binaryValueToTest := ADR(valueToTest);
assertionIsWrong := (binaryValueToTest^ <> THIS^.BINARY_NEGATIVE_INFINITY);

message := SEL(
	assertionIsWrong,
	'currentValue is %s assertion must be TRUE', 
	'currentValue is %s assertion must be FALSE'
);

valueToTestAsString := TO_STRING(valueToTest);

messageStringBuilder(
	sFormat := message,
	arg1 := THIS^.AnyToArg(valueToTestAsString)
);

THIS^.assertorContainer.assertor.assert.float.single.valueIsNegativeInfinite(
	currentValue := valueToTest,
	message := ''
);

THIS^.AssertEquals_BOOL(
	Expected 	:= assertionIsWrong,
	Actual 		:= THIS^.assertorContainer.wasAssertionWrong,
	Message 	:= messageStringBuilder.sOut
);
END_METHOD

(*

short summary
==================
This test method tests ``assert.float.single.valueIsNegativeZero``
method of CNM_AssertionInterfaces library, 
it provides the possibility to handover test data via parameter 

.. <legal notes>

legal notes
=================
| SPDX-FileCopyrightText: © 2022 ekvip automation GmbH <info@ekvip.de>
| SPDX-License-Identifier: Apache-2.0
| For details check: Apache-2.0_

.. _Apache-2.0: https://www.apache.org/licenses/LICENSE-2.0

.. </legal notes>

parameters
==========

*)

METHOD testValueIsNegativeZero
VAR_INPUT
	(* for the test it's the parameter ``currentValue`` *)
	valueToTest	:REAL;	
END_VAR
VAR
	(* just the expectation if the assertion to test must be worng or true *)
	assertionIsWrong		:BOOL;
	(* contains the format string for the test message *)
	message					:Tc2_System.T_MaxString;
	(* TwinCAT printf with the test message *)
	messageStringBuilder	:Tc2_Utilities.FB_FormatString;
	(* value of the paramter ``valueToTest`` as string *)
	valueToTestAsString		:Tc2_System.T_MaxString;
	(* binary value of the parameter ``valueToTest`` *)
	binaryValueToTest		:POINTER TO DWORD;
	(* sgin bit as BYTE for the message *)
	signBitAsByte			:BYTE;
	(* sgin bit as BOOL for the message *)
	signBit					:BOOL;	
END_VAR
THIS^.assertorContainer.resetAssertor();

binaryValueToTest := ADR(valueToTest);
signBit := binaryValueToTest^.SIGN;
signBitAsByte := TO_BYTE(signBit);

assertionIsWrong := (binaryValueToTest^ <> THIS^.BINARY_MINUS_ZERO);

message := SEL(
	assertionIsWrong,
	'currentValue is %s and sign bit is %u assertion must be TRUE', 
	'currentValue is %s and sign bit is %u assertion must be FALSE'
);

valueToTestAsString := TO_STRING(valueToTest);

messageStringBuilder(
	sFormat := message,
	arg1 := THIS^.AnyToArg(valueToTestAsString),
	arg2 := THIS^.AnyToArg(signBitAsByte)
);

THIS^.assertorContainer.assertor.assert.float.single.valueIsNegativeZero(
	currentValue := valueToTest,
	message := ''
);

THIS^.AssertEquals_BOOL(
	Expected 	:= assertionIsWrong,
	Actual 		:= THIS^.assertorContainer.wasAssertionWrong,
	Message 	:= messageStringBuilder.sOut
);
END_METHOD

(*

short summary
==================
This test method tests ``assert.float.single.valueIsNormal``
method of CNM_AssertionInterfaces library, 
it provides the possibility to handover test data via parameter 

.. <legal notes>

legal notes
=================
| SPDX-FileCopyrightText: © 2022 ekvip automation GmbH <info@ekvip.de>
| SPDX-License-Identifier: Apache-2.0
| For details check: Apache-2.0_

.. _Apache-2.0: https://www.apache.org/licenses/LICENSE-2.0

.. </legal notes>

parameters
==========

*)

METHOD testValueIsNormal
VAR_INPUT
	(* for the test it's the parameter ``currentValue`` *)
	valueToTest	:REAL;	
END_VAR
VAR
	(* just the expectation if the assertion to test must be worng or true *)
	assertionIsWrong		:BOOL;
	(* contains the format string for the test message *)
	message					:Tc2_System.T_MaxString;
	(* TwinCAT printf with the test message *)
	messageStringBuilder	:Tc2_Utilities.FB_FormatString;
	(* value of the paramter ``valueToTest`` as string *)
	valueToTestAsString		:Tc2_System.T_MaxString;
	(* binary value of the parameter ``valueToTest`` *)
	binaryValueToTest		:POINTER TO DWORD;
END_VAR
THIS^.assertorContainer.resetAssertor();

binaryValueToTest := ADR(valueToTest);

assertionIsWrong := (
	((binaryValueToTest^ AND THIS^.MASK_FOR_EXPONENT) = THIS^.BINARY_ZERO)
	OR_ELSE Tc2_Utilities.RealIsNaN(valueToTest)
	OR_ELSE (NOT Tc2_Utilities.RealIsFinite(valueToTest))
);

message := SEL(
	assertionIsWrong,
	'currentValue is %s assertion must be TRUE', 
	'currentValue is %s assertion must be FALSE'
);

valueToTestAsString := TO_STRING(valueToTest);

messageStringBuilder(
	sFormat := message,
	arg1 := THIS^.AnyToArg(valueToTestAsString)
);

THIS^.assertorContainer.assertor.assert.float.single.valueIsNormal(
	currentValue := valueToTest,
	message := ''
);

THIS^.AssertEquals_BOOL(
	Expected 	:= assertionIsWrong,
	Actual 		:= THIS^.assertorContainer.wasAssertionWrong,
	Message 	:= messageStringBuilder.sOut
);
END_METHOD

(*

short summary
==================
This test method tests ``assert.float.single.valueIsNotEqualTo``
method of CNM_AssertionInterfaces library, 
it provides the possibility to handover test data via parameter 


.. <legal notes>

legal notes
=================
| SPDX-FileCopyrightText: © 2022 ekvip automation GmbH <info@ekvip.de>
| SPDX-License-Identifier: Apache-2.0
| For details check: Apache-2.0_

.. _Apache-2.0: https://www.apache.org/licenses/LICENSE-2.0

.. </legal notes>

parameters
==========

*)

METHOD testValueIsNotEqualTo 
VAR_INPUT
	(* for the test it's the parameter ``currentValue`` *)
	valueToTest		:REAL;
	(* for the test it's the parameter ``unexpectedValue`` *)
	unexpectedValue	:REAL;
	(* for the test it's the parameter ``tolerance`` *)
	tolerance		:REAL;
END_VAR
VAR
	(* just the expectation if the assertion to test must be worng or true *)
	assertionIsWrong		:BOOL;
	(* contains the format string for the test message *)
	message					:Tc2_System.T_MaxString;
	(* TwinCAT printf with the test message *)
	messageStringBuilder	:Tc2_Utilities.FB_FormatString;
	(* just to cast *)
	binaryCurrentValue		:POINTER TO DWORD;
	(* just to cast *)
	binaryUnexpectedValue	:POINTER TO DWORD;
	(* value of the paramter ``valueToTest`` as string *)
	valueToTestAsString		:Tc2_System.T_MaxString;
	(* value of the paramter ``unexpectedValue`` as string *)
	unexpectedValueAsString	:Tc2_System.T_MaxString;
	(* value of the paramter ``tolerance`` as string *)
	toleranceAsString		:Tc2_System.T_MaxString;	
END_VAR
THIS^.assertorContainer.resetAssertor();
IF (
	Tc2_Utilities.RealIsNaN(valueToTest)
	OR Tc2_Utilities.RealIsNaN(unexpectedValue)
	OR Tc2_Utilities.RealIsNaN(tolerance)
) THEN
	assertionIsWrong := FALSE;
ELSIF (NOT Tc2_Utilities.RealIsFinite(tolerance)) THEN
	assertionIsWrong := TRUE;
ELSIF (Tc2_Utilities.RealIsFinite(valueToTest) <> Tc2_Utilities.RealIsFinite(unexpectedValue)) THEN
	assertionIsWrong := FALSE; 
ELSIF (
	(NOT Tc2_Utilities.RealIsFinite(valueToTest))
	OR (NOT Tc2_Utilities.RealIsFinite(unexpectedValue))
) THEN
	binaryCurrentValue := ADR(valueToTest);
	binaryUnexpectedValue := ADR(unexpectedValue);
	assertionIsWrong := (binaryCurrentValue^.SIGN = binaryUnexpectedValue^.SIGN);
ELSE
	assertionIsWrong := (
		((unexpectedValue + ABS(tolerance)) >= valueToTest)
		AND ((unexpectedValue - ABS(tolerance)) <= valueToTest)
	);
END_IF

message := SEL(
	assertionIsWrong,
	'currentValue is %s unexpectedValue is %s tolerance is %s assertion must be TRUE', 
	'currentValue is %s unexpectedValue is %s tolerance is %s assertion must be FALSE'
);

valueToTestAsString := TO_STRING(valueToTest);
unexpectedValueAsString := TO_STRING(unexpectedValue);
toleranceAsString := TO_STRING(tolerance);

messageStringBuilder(
	sFormat := message,
	arg1 := THIS^.AnyToArg(valueToTestAsString),
	arg2 := THIS^.AnyToArg(unexpectedValueAsString),
	arg3 := THIS^.AnyToArg(toleranceAsString)
);

THIS^.assertorContainer.assertor.assert.float.single.valueIsNotEqualTo(
	currentValue	:= valueToTest,
	unexpectedValue	:= unexpectedValue,
	tolerance       := tolerance,
	message			:= ''
);

THIS^.AssertEquals_BOOL(
	Expected 	:= assertionIsWrong,
	Actual 		:= THIS^.assertorContainer.wasAssertionWrong,
	Message 	:= messageStringBuilder.sOut
);
END_METHOD

(*

short summary
==================
This test method tests ``assert.float.single.valueIsNotNegativeInfinite``
method of CNM_AssertionInterfaces library, 
it provides the possibility to handover test data via parameter 

.. <legal notes>

legal notes
=================
| SPDX-FileCopyrightText: © 2022 ekvip automation GmbH <info@ekvip.de>
| SPDX-License-Identifier: Apache-2.0
| For details check: Apache-2.0_

.. _Apache-2.0: https://www.apache.org/licenses/LICENSE-2.0

.. </legal notes>

parameters
==========

*)

METHOD testValueIsNotNegativeInfinite
VAR_INPUT
	(* for the test it's the parameter ``currentValue`` *)
	valueToTest	:REAL;	
END_VAR
VAR
	(* just the expectation if the assertion to test must be worng or true *)
	assertionIsWrong		:BOOL;
	(* contains the format string for the test message *)
	message					:Tc2_System.T_MaxString;
	(* TwinCAT printf with the test message *)
	messageStringBuilder	:Tc2_Utilities.FB_FormatString;
	(* value of the paramter ``valueToTest`` as string *)
	valueToTestAsString		:Tc2_System.T_MaxString;
	(* binary value of the parameter ``valueToTest`` *)
	binaryValueToTest		:POINTER TO DWORD;
END_VAR
THIS^.assertorContainer.resetAssertor();

binaryValueToTest := ADR(valueToTest);
assertionIsWrong := (binaryValueToTest^ = THIS^.BINARY_NEGATIVE_INFINITY);

message := SEL(
	assertionIsWrong,
	'currentValue is %s assertion must be TRUE', 
	'currentValue is %s assertion must be FALSE'
);

valueToTestAsString := TO_STRING(valueToTest);

messageStringBuilder(
	sFormat := message,
	arg1 := THIS^.AnyToArg(valueToTestAsString)
);

THIS^.assertorContainer.assertor.assert.float.single.valueIsNotNegativeInfinite(
	currentValue := valueToTest,
	message := ''
);

THIS^.AssertEquals_BOOL(
	Expected 	:= assertionIsWrong,
	Actual 		:= THIS^.assertorContainer.wasAssertionWrong,
	Message 	:= messageStringBuilder.sOut
);
END_METHOD

(*

short summary
==================
This test method tests ``assert.float.single.valueIsNotPositiveInfinite``
method of CNM_AssertionInterfaces library, 
it provides the possibility to handover test data via parameter 

.. <legal notes>

legal notes
=================
| SPDX-FileCopyrightText: © 2022 ekvip automation GmbH <info@ekvip.de>
| SPDX-License-Identifier: Apache-2.0
| For details check: Apache-2.0_

.. _Apache-2.0: https://www.apache.org/licenses/LICENSE-2.0

.. </legal notes>

parameters
==========

*)

METHOD testValueIsNotPositiveInfinite
VAR_INPUT
	(* for the test it's the parameter ``currentValue`` *)
	valueToTest	:REAL;	
END_VAR
VAR
	(* just the expectation if the assertion to test must be worng or true *)
	assertionIsWrong		:BOOL;
	(* contains the format string for the test message *)
	message					:Tc2_System.T_MaxString;
	(* TwinCAT printf with the test message *)
	messageStringBuilder	:Tc2_Utilities.FB_FormatString;
	(* value of the paramter ``valueToTest`` as string *)
	valueToTestAsString		:Tc2_System.T_MaxString;
	(* binary value of the parameter ``valueToTest`` *)
	binaryValueToTest		:POINTER TO DWORD;
END_VAR
THIS^.assertorContainer.resetAssertor();

binaryValueToTest := ADR(valueToTest);
assertionIsWrong := (binaryValueToTest^ = THIS^.BINARY_INFINITY);

message := SEL(
	assertionIsWrong,
	'currentValue is %s assertion must be TRUE', 
	'currentValue is %s assertion must be FALSE'
);

valueToTestAsString := TO_STRING(valueToTest);

messageStringBuilder(
	sFormat := message,
	arg1 := THIS^.AnyToArg(valueToTestAsString)
);

THIS^.assertorContainer.assertor.assert.float.single.valueIsNotPositiveInfinite(
	currentValue := valueToTest,
	message := ''
);

THIS^.AssertEquals_BOOL(
	Expected 	:= assertionIsWrong,
	Actual 		:= THIS^.assertorContainer.wasAssertionWrong,
	Message 	:= messageStringBuilder.sOut
);
END_METHOD

(*

short summary
==================
This test method tests ``assert.float.single.valueIsNotSpecial``
method of CNM_AssertionInterfaces library, 
it provides the possibility to handover test data via parameter 

.. <legal notes>

legal notes
=================
| SPDX-FileCopyrightText: © 2022 ekvip automation GmbH <info@ekvip.de>
| SPDX-License-Identifier: Apache-2.0
| For details check: Apache-2.0_

.. _Apache-2.0: https://www.apache.org/licenses/LICENSE-2.0

.. </legal notes>

parameters
==========

*)

METHOD testValueIsNotSpecial
VAR_INPUT
	(* for the test it's the parameter ``currentValue`` *)
	valueToTest	:REAL;	
END_VAR
VAR
	(* just the expectation if the assertion to test must be worng or true *)
	assertionIsWrong		:BOOL;
	(* contains the format string for the test message *)
	message					:Tc2_System.T_MaxString;
	(* TwinCAT printf with the test message *)
	messageStringBuilder	:Tc2_Utilities.FB_FormatString;
	(* value of the paramter ``valueToTest`` as string *)
	valueToTestAsString		:Tc2_System.T_MaxString;
END_VAR
THIS^.assertorContainer.resetAssertor();

assertionIsWrong := (
	(NOT Tc2_Utilities.RealIsFinite(valueToTest))
	OR_ELSE Tc2_Utilities.RealIsNaN(valueToTest)
);

message := SEL(
	assertionIsWrong,
	'currentValue is %s assertion must be TRUE', 
	'currentValue is %s assertion must be FALSE'
);

valueToTestAsString := TO_STRING(valueToTest);

messageStringBuilder(
	sFormat := message,
	arg1 := THIS^.AnyToArg(valueToTestAsString)
);

THIS^.assertorContainer.assertor.assert.float.single.valueIsNotSpecial(
	currentValue := valueToTest,
	message := ''
);

THIS^.AssertEquals_BOOL(
	Expected 	:= assertionIsWrong,
	Actual 		:= THIS^.assertorContainer.wasAssertionWrong,
	Message 	:= messageStringBuilder.sOut
);
END_METHOD

(*

short summary
==================
This test method tests ``assert.float.single.valueIsPositive``
method of CNM_AssertionInterfaces library, 
it provides the possibility to handover test data via parameter 

.. <legal notes>

legal notes
=================
| SPDX-FileCopyrightText: © 2022 ekvip automation GmbH <info@ekvip.de>
| SPDX-License-Identifier: Apache-2.0
| For details check: Apache-2.0_

.. _Apache-2.0: https://www.apache.org/licenses/LICENSE-2.0

.. </legal notes>

parameters
==========

*)

METHOD testValueIsPositive
VAR_INPUT
	(* for the test it's the parameter ``currentValue`` *)
	valueToTest	:REAL;	
END_VAR
VAR
	(* just the expectation if the assertion to test must be worng or true *)
	assertionIsWrong		:BOOL;
	(* contains the format string for the test message *)
	message					:Tc2_System.T_MaxString;
	(* TwinCAT printf with the test message *)
	messageStringBuilder	:Tc2_Utilities.FB_FormatString;
	(* value of the paramter ``valueToTest`` as string *)
	valueToTestAsString		:Tc2_System.T_MaxString;
	(* binary value of the parameter ``valueToTest`` *)
	binaryValueToTest		:POINTER TO DWORD;
	(* sgin bit as BYTE for the message *)
	signBitAsByte			:BYTE;
	(* sgin bit as BOOL for the message *)
	signBit					:BOOL;	
END_VAR
THIS^.assertorContainer.resetAssertor();

binaryValueToTest := ADR(valueToTest);
signBit := binaryValueToTest^.SIGN;
signBitAsByte := TO_BYTE(signBit);
assertionIsWrong := (
	signBit
	OR Tc2_Utilities.RealIsNaN(valueToTest)
);

message := SEL(
	assertionIsWrong,
	'currentValue is %s and sign bit is %u assertion must be TRUE', 
	'currentValue is %s and sign bit is %u assertion must be FALSE'
);

valueToTestAsString := TO_STRING(valueToTest);

messageStringBuilder(
	sFormat := message,
	arg1 := THIS^.AnyToArg(valueToTestAsString),
	arg2 := THIS^.AnyToArg(signBitAsByte)
);

THIS^.assertorContainer.assertor.assert.float.single.valueIsPositive(
	currentValue := valueToTest,
	message := ''
);

THIS^.AssertEquals_BOOL(
	Expected 	:= assertionIsWrong,
	Actual 		:= THIS^.assertorContainer.wasAssertionWrong,
	Message 	:= messageStringBuilder.sOut
);
END_METHOD

(*

short summary
==================
This test method tests ``assert.float.single.valueIsPositiveInfinite``
method of CNM_AssertionInterfaces library, 
it provides the possibility to handover test data via parameter 

.. <legal notes>

legal notes
=================
| SPDX-FileCopyrightText: © 2022 ekvip automation GmbH <info@ekvip.de>
| SPDX-License-Identifier: Apache-2.0
| For details check: Apache-2.0_

.. _Apache-2.0: https://www.apache.org/licenses/LICENSE-2.0

.. </legal notes>

parameters
==========

*)

METHOD testValueIsPositiveInfinite
VAR_INPUT
	(* for the test it's the parameter ``currentValue`` *)
	valueToTest	:REAL;	
END_VAR
VAR
	(* just the expectation if the assertion to test must be worng or true *)
	assertionIsWrong		:BOOL;
	(* contains the format string for the test message *)
	message					:Tc2_System.T_MaxString;
	(* TwinCAT printf with the test message *)
	messageStringBuilder	:Tc2_Utilities.FB_FormatString;
	(* value of the paramter ``valueToTest`` as string *)
	valueToTestAsString		:Tc2_System.T_MaxString;
	(* binary value of the parameter ``valueToTest`` *)
	binaryValueToTest		:POINTER TO DWORD;
END_VAR
THIS^.assertorContainer.resetAssertor();

binaryValueToTest := ADR(valueToTest);
assertionIsWrong := (binaryValueToTest^ <> THIS^.BINARY_INFINITY);

message := SEL(
	assertionIsWrong,
	'currentValue is %s assertion must be TRUE', 
	'currentValue is %s assertion must be FALSE'
);

valueToTestAsString := TO_STRING(valueToTest);

messageStringBuilder(
	sFormat := message,
	arg1 := THIS^.AnyToArg(valueToTestAsString)
);

THIS^.assertorContainer.assertor.assert.float.single.valueIsPositiveInfinite(
	currentValue := valueToTest,
	message := ''
);

THIS^.AssertEquals_BOOL(
	Expected 	:= assertionIsWrong,
	Actual 		:= THIS^.assertorContainer.wasAssertionWrong,
	Message 	:= messageStringBuilder.sOut
);
END_METHOD

(*

short summary
==================
This test method tests ``assert.float.single.valueIsPositiveZero``
method of CNM_AssertionInterfaces library, 
it provides the possibility to handover test data via parameter 

.. <legal notes>

legal notes
=================
| SPDX-FileCopyrightText: © 2022 ekvip automation GmbH <info@ekvip.de>
| SPDX-License-Identifier: Apache-2.0
| For details check: Apache-2.0_

.. _Apache-2.0: https://www.apache.org/licenses/LICENSE-2.0

.. </legal notes>

parameters
==========

*)

METHOD testValueIsPositiveZero
VAR_INPUT
	(* for the test it's the parameter ``currentValue`` *)
	valueToTest	:REAL;	
END_VAR
VAR
	(* just the expectation if the assertion to test must be worng or true *)
	assertionIsWrong		:BOOL;
	(* contains the format string for the test message *)
	message					:Tc2_System.T_MaxString;
	(* TwinCAT printf with the test message *)
	messageStringBuilder	:Tc2_Utilities.FB_FormatString;
	(* value of the paramter ``valueToTest`` as string *)
	valueToTestAsString		:Tc2_System.T_MaxString;
	(* binary value of the parameter ``valueToTest`` *)
	binaryValueToTest		:POINTER TO DWORD;
	(* sgin bit as BYTE for the message *)
	signBitAsByte			:BYTE;
	(* sgin bit as BOOL for the message *)
	signBit					:BOOL;	
END_VAR
THIS^.assertorContainer.resetAssertor();

binaryValueToTest := ADR(valueToTest);
signBit := binaryValueToTest^.SIGN;
signBitAsByte := TO_BYTE(signBit);

assertionIsWrong := (binaryValueToTest^ <> THIS^.BINARY_ZERO);

message := SEL(
	assertionIsWrong,
	'currentValue is %s and sign bit is %u assertion must be TRUE', 
	'currentValue is %s and sign bit is %u assertion must be FALSE'
);

valueToTestAsString := TO_STRING(valueToTest);

messageStringBuilder(
	sFormat := message,
	arg1 := THIS^.AnyToArg(valueToTestAsString),
	arg2 := THIS^.AnyToArg(signBitAsByte)
);

THIS^.assertorContainer.assertor.assert.float.single.valueIsPositiveZero(
	currentValue := valueToTest,
	message := ''
);

THIS^.AssertEquals_BOOL(
	Expected 	:= assertionIsWrong,
	Actual 		:= THIS^.assertorContainer.wasAssertionWrong,
	Message 	:= messageStringBuilder.sOut
);
END_METHOD

(*

short summary
==================
This test method tests ``assert.float.single.valueIsSpecial``
method of CNM_AssertionInterfaces library, 
it provides the possibility to handover test data via parameter 

.. <legal notes>

legal notes
=================
| SPDX-FileCopyrightText: © 2022 ekvip automation GmbH <info@ekvip.de>
| SPDX-License-Identifier: Apache-2.0
| For details check: Apache-2.0_

.. _Apache-2.0: https://www.apache.org/licenses/LICENSE-2.0

.. </legal notes>

parameters
==========

*)

METHOD testValueIsSpecial
VAR_INPUT
	(* for the test it's the parameter ``currentValue`` *)
	valueToTest	:REAL;	
END_VAR
VAR
	(* just the expectation if the assertion to test must be worng or true *)
	assertionIsWrong		:BOOL;
	(* contains the format string for the test message *)
	message					:Tc2_System.T_MaxString;
	(* TwinCAT printf with the test message *)
	messageStringBuilder	:Tc2_Utilities.FB_FormatString;
	(* value of the paramter ``valueToTest`` as string *)
	valueToTestAsString		:Tc2_System.T_MaxString;
END_VAR
THIS^.assertorContainer.resetAssertor();

assertionIsWrong := (
	Tc2_Utilities.RealIsFinite(valueToTest)
	AND_THEN (NOT Tc2_Utilities.RealIsNaN(valueToTest))
);

message := SEL(
	assertionIsWrong,
	'currentValue is %s assertion must be TRUE', 
	'currentValue is %s assertion must be FALSE'
);

valueToTestAsString := TO_STRING(valueToTest);

messageStringBuilder(
	sFormat := message,
	arg1 := THIS^.AnyToArg(valueToTestAsString)
);

THIS^.assertorContainer.assertor.assert.float.single.valueIsSpecial(
	currentValue := valueToTest,
	message := ''
);

THIS^.AssertEquals_BOOL(
	Expected 	:= assertionIsWrong,
	Actual 		:= THIS^.assertorContainer.wasAssertionWrong,
	Message 	:= messageStringBuilder.sOut
);
END_METHOD

(*

short summary
==================
This test method tests ``assert.float.single.valueIsSubnormal``
method of CNM_AssertionInterfaces library, 
it provides the possibility to handover test data via parameter 

.. <legal notes>

legal notes
=================
| SPDX-FileCopyrightText: © 2022 ekvip automation GmbH <info@ekvip.de>
| SPDX-License-Identifier: Apache-2.0
| For details check: Apache-2.0_

.. _Apache-2.0: https://www.apache.org/licenses/LICENSE-2.0

.. </legal notes>

parameters
==========

*)

METHOD testValueIsSubnormal
VAR_INPUT
	(* for the test it's the parameter ``currentValue`` *)
	valueToTest	:REAL;	
END_VAR
VAR
	(* just the expectation if the assertion to test must be worng or true *)
	assertionIsWrong		:BOOL;
	(* contains the format string for the test message *)
	message					:Tc2_System.T_MaxString;
	(* TwinCAT printf with the test message *)
	messageStringBuilder	:Tc2_Utilities.FB_FormatString;
	(* value of the paramter ``valueToTest`` as string *)
	valueToTestAsString		:Tc2_System.T_MaxString;
	(* binary value of the parameter ``valueToTest`` *)
	binaryValueToTest		:POINTER TO DWORD;
END_VAR
THIS^.assertorContainer.resetAssertor();

binaryValueToTest := ADR(valueToTest);

assertionIsWrong := (
	((binaryValueToTest^ AND THIS^.MASK_FOR_EXPONENT) <> THIS^.BINARY_ZERO)
);

message := SEL(
	assertionIsWrong,
	'currentValue is %s assertion must be TRUE', 
	'currentValue is %s assertion must be FALSE'
);

valueToTestAsString := TO_STRING(valueToTest);

messageStringBuilder(
	sFormat := message,
	arg1 := THIS^.AnyToArg(valueToTestAsString)
);

THIS^.assertorContainer.assertor.assert.float.single.valueIsSubnormal(
	currentValue := valueToTest,
	message := ''
);

THIS^.AssertEquals_BOOL(
	Expected 	:= assertionIsWrong,
	Actual 		:= THIS^.assertorContainer.wasAssertionWrong,
	Message 	:= messageStringBuilder.sOut
);
END_METHOD

END_FUNCTION_BLOCK

(* stored: Version 1.1.0.1, ProductVersion 3.1.4026.13
   POU RealAssertionTests: Id {e23c241e-ac94-4686-844e-ef6a5b49b964}, SpecialFunc None
   Folder internal: Id {cea34b2b-f8cd-415e-90b6-44170d1fb25e}
   Folder valueIsANumber: Id {89e2fefa-f021-4acd-b88f-3ba0580535c9}
   Folder valueIsEqualTo: Id {c8ef93a6-9921-4921-9085-8816d2df969d}
   Folder valueIsFinite: Id {053d53e2-d311-4927-bf21-d1f017979f9c}
   Folder valueIsGreaterThan: Id {c00bb4fc-e9e0-484b-916b-856bad594b5e}
   Folder valueIsInfinite: Id {598dd276-7497-4077-bc1b-98ae0390a85a}
   Folder valueIsInRangeOf: Id {62434e16-e11c-4a3f-a29d-22d3c26a3bab}
   Folder valueIsLessThan: Id {3de12dba-d8ea-4413-a2bb-e6771356dd0c}
   Folder valueIsMax: Id {cf6aa9ec-1954-405d-83e3-2331d5ac7e04}
   Folder valueIsMin: Id {9c679ce5-2a7a-428a-9488-6c09d21e003b}
   Folder valueIsNaN: Id {6eda3375-157a-49cb-bf59-8e4319affb62}
   Folder valueIsNegative: Id {851965bc-1f59-4aad-92bc-4468a72795b3}
   Folder valueIsNegativeInfinite: Id {580720b3-4b87-44e3-9e01-abba4c01f78a}
   Folder valueIsNegativeZero: Id {7511257b-98ef-4ac4-b8ad-af8ab9b980c4}
   Folder valueIsNormal: Id {0cf3bd59-a845-4cd4-b9c5-7e1826c6f37e}
   Folder valueIsNotEqualTo: Id {f51f5dfb-d0b3-4728-8e55-1bf8af1a8f7f}
   Folder valueIsNotNegativeInfinite: Id {b7d72bc2-232f-41cb-878a-17ee405dafef}
   Folder valueIsNotPositiveInfinite: Id {291f9f79-287d-401f-85d0-fe95adc2ff4b}
   Folder valueIsNotSpecial: Id {231f0e2f-845c-4e7e-8dfb-be5119a7ff02}
   Folder valueIsPositive: Id {d9b7df8e-3e15-4dcd-81d1-10adca8db28d}
   Folder valueIsPositiveInfinite: Id {635c1f31-d0fb-4150-9f3f-c4f80c670fe6}
   Folder valueIsPositiveZero: Id {e5627c44-1d82-4bf1-8bd1-a279b7506530}
   Folder valueIsSpecial: Id {75ea6933-bf55-4d30-9d72-2afbba19f344}
   Folder valueIsSubnormal: Id {515b5c9e-1c3b-4b6a-bc56-f4c194a70c56}
   Method FB_init: Id {9c998664-6110-496c-87ec-0518d2070d66}
   Method getTestNameFor: Id {beb963f5-55c0-404d-81ce-8eee3fcfa33b}
   Method runValueIsANumberTests: Id {a17b9a36-dc78-44e4-b520-2939338bd828}
   Method runValueIsEqualToTests: Id {5fb805db-473f-408c-b918-5b1a6c1ff7b6}
   Method runValueIsFiniteTests: Id {2066167f-8676-46c8-9900-59b321470bbb}
   Method runValueIsGreaterThanTests: Id {004c54d7-7922-452e-b6ad-4e6eb7dfef0f}
   Method runValueIsInfiniteTests: Id {d772de01-9962-4a94-ae36-ee27a0d1603b}
   Method runValueIsInRangeOfTests: Id {457e2119-5278-402b-9b44-8a3d62f9299d}
   Method runValueIsLessThanTests: Id {744fb4a7-de68-4cec-a87e-f720f59f9683}
   Method runValueIsMaxTests: Id {5c7b8d96-3401-4b4c-9cc1-1a4d8495dfc1}
   Method runValueIsMinTests: Id {83dcc8f2-9a14-4a17-9d35-47566af65af8}
   Method runValueIsNaNTests: Id {663360d1-a84c-4cc8-987b-458ea3d46db1}
   Method runValueIsNegativeInfiniteTests: Id {56b01109-422e-46d1-95d4-290b7e86882b}
   Method runValueIsNegativeTests: Id {887e219f-0f1e-4ceb-bdbb-01b48efb24b1}
   Method runValueIsNegativeZeroTests: Id {cffae337-3f18-4e05-925d-b4ca6668b3a0}
   Method runValueIsNormalTests: Id {bdb7a2a4-4ffa-44b8-9301-e045c8b02163}
   Method runValueIsNotEqualToTests: Id {fc0d1cb8-e9bb-42e5-bf62-649768306731}
   Method runValueIsNotNegativeInfiniteTests: Id {315e317a-afff-4a59-abd6-d60fc470fca3}
   Method runValueIsNotPositiveInfiniteTests: Id {a5e23a78-1ba5-43f5-9f53-ad430a80b03a}
   Method runValueIsNotSpecialTests: Id {042931ad-8fa7-46d3-915b-4151ce3d9580}
   Method runValueIsPositiveInfiniteTests: Id {6511d732-7643-4cde-a606-ab11efa7b06c}
   Method runValueIsPositiveTests: Id {369045cc-0df3-488c-bab0-633ac95508f7}
   Method runValueIsPositiveZeroTests: Id {ec38ec20-afd1-4bc2-a2a0-bf7aec76c460}
   Method runValueIsSpecialTests: Id {46f5e997-c1f5-40bf-a67a-c2dc7e1e14c6}
   Method runValueIsSubnormalTests: Id {331144eb-b692-4a79-af4b-321b35aa9d8f}
   Method testValueIsANumber: Id {9169311a-cfa6-4e6d-955b-85779031daab}
   Method testValueIsEqualTo: Id {e17dbc53-0252-4af6-a5ce-689d522a75b5}
   Method testValueIsFinite: Id {9fe48ce8-cad6-46fb-99b1-735c4cf302ff}
   Method testValueIsGreaterThan: Id {03c1e3c7-00ad-4238-85e5-efc3e1727906}
   Method testValueIsInfinite: Id {22fcab4f-58f7-4eb7-b997-2d3c57087c34}
   Method testValueIsInRangeOf: Id {282b6902-46bc-490c-a423-131e67af79e2}
   Method testValueIsLessThan: Id {30539b72-a02c-4994-a9a8-52392731ff71}
   Method testValueIsMax: Id {c8193b8c-c571-40fb-8887-e6e1df6f33e3}
   Method testValueIsMin: Id {eb605393-b37d-4989-80e8-20787e0228a9}
   Method testValueIsNaN: Id {73123b70-48e2-4748-9014-7077af7d43a3}
   Method testValueIsNegative: Id {3f36264b-8058-43aa-8080-967b493e92b0}
   Method testValueIsNegativeInfinite: Id {792c88d0-1fcc-4837-b9e9-d415d91e7d36}
   Method testValueIsNegativeZero: Id {35815cc5-cf64-4322-b68c-05812318751b}
   Method testValueIsNormal: Id {3059db8d-98a4-47a6-9c40-8d713db3b5b8}
   Method testValueIsNotEqualTo: Id {009f2fe4-8b85-4124-8a32-e2cb219762cc}
   Method testValueIsNotNegativeInfinite: Id {b101570c-dfa4-4b97-aa7e-dc019fb96b33}
   Method testValueIsNotPositiveInfinite: Id {f321642f-d04c-4fd8-ab40-cee9728af8bc}
   Method testValueIsNotSpecial: Id {b0e3018a-452e-43ee-947b-9f4952ded9f6}
   Method testValueIsPositive: Id {d3a9d5ca-38b1-4455-9196-090179b6fd44}
   Method testValueIsPositiveInfinite: Id {8eecd20e-674f-4873-8156-3763d31ea329}
   Method testValueIsPositiveZero: Id {d52e5ab6-bfa1-436d-857a-dc1038fd8ae8}
   Method testValueIsSpecial: Id {97139f36-742e-4105-ad18-87e158a000cd}
   Method testValueIsSubnormal: Id {1df82d4f-0dd4-48c1-bccd-cadaa0ece362} *)
